# B&R Automation Studio project NAEUL004C00R13L518F00 (part 67)

#### Act_InitGlobal.st - Change By Project
```iecst
(** 2019-04-16 **)
ACTION Act_InitGlobal:

	(* Always Change If Project Change *)

	//Pass Data To Link

	p_bLinkNtParamMagConv1Prep ACCESS p_NtParamProjMag1ConvPrep;
	p_bLinkNtParamMagConv2Prep ACCESS p_NtParamProjMag2ConvPrep;
	p_bLinkNtParamMagConv3Prep ACCESS p_NtParamProjMag3ConvPrep;
	p_bLinkUSHermesABlkUS ACCESS p_USHermesABlkUS;
	p_bLinkUSHermesBBlkUS ACCESS p_USHermesBBlkUS;
	p_bLinkFollower1USAllow ACCESS p_Follower1USAllow;
	p_bLinkFollower2DSAllow ACCESS p_Follower2DSAllow;
	p_bLinkProjLifterMagPlatform ACCESS p_NtParamProjLifterMagPlatform;
	p_bLinkDIPshrAntiJamSen ACCESS p_DIPshrAntiJamSen;
	p_bLinkCurtainSen ACCESS p_DICurtainSen;
	p_bLinkPshrRetSen ACCESS p_DIPusherRetRS;

	p_diBuffer1NxtLoadSlt ACCESS p_Buffer1NxtLoadSlt;
	p_diBuffer2NxtLoadSlt ACCESS p_Buffer2NxtLoadSlt;
	p_diBuffer3NxtLoadSlt ACCESS p_Buffer3NxtLoadSlt;

	p_diMinSlt ACCESS p_ProdRcpCurrRcp1MinSltValue;
	p_diMaxSlt ACCESS p_ProdRcpCurrRcp1MaxSltValue;

	p_bTopToBtm ACCESS p_ProdRcpCurrRcp1TopToBtm;

	p_bLinkMcParamMagWidthChkDis ACCESS p_McParamMagWidthChkDis;

	//p_bMagWidthChkDis
	p_sLinkProdRcpCurrRcp1Nm ACCESS p_ProdRcpCurrRcp1Nm;
	p_diLinkProdRcpCurrRcp1Pitch ACCESS p_ProdRcpCurrRcp1Pitch;
	p_sLinkMagRcpCurrRcpNm ACCESS p_MagRcpCurrRcpNm;

	//Pass Data To Internal Use
	p_udiRstErr ACCESS p_RstErrReset;
	p_bRun ACCESS p_OpsRun;
	p_bStop ACCESS p_OpsStop;
	p_bStep ACCESS p_OpsStep;

	p_tShutterWaitTmr ACCESS p_NtParamShutterWaitTmr;
	p_bCurtainSenPrep ACCESS p_NtParamCurtainSenPrep;

	p_sProgNm ACCESS p_NtParamOpsTravLifULProgNm;
	p_bNtSettingsLoadDone ACCESS p_StartupNtSettingsLoadDone;

	p_eULMag ACCESS p_NtParamProjMag;
	p_bInShutDis ACCESS p_McParamInShutterDis;

	p_eUSCommMod1 ACCESS p_McParamUSCommAMod;
	p_eUSCommMod2 ACCESS p_McParamUSCommBMod;

	p_eUSSMEMAStat1 ACCESS p_USSMEMAAStat;
	p_eUSSMEMAStatus1 ACCESS p_USSMEMAAStatus;
	p_bUSSMEMAUSRdy1 ACCESS p_USSMEMAAUSRdy;
	p_bUSSMEMAGdBrdRdy1 ACCESS p_USSMEMAAUSGdBrdRdy;
	p_bUSSMEMATransporting1 ACCESS p_USSMEMAATransporting;
	p_bUSSMEMAConvStart1 ACCESS p_USSMEMAAConvStart;
	p_bUSSMEMAConvStop1 ACCESS p_USSMEMAAConvStop;

	p_eUSSMEMAStat2 ACCESS p_USSMEMABStat;
	p_eUSSMEMAStatus2 ACCESS p_USSMEMABStatus;
	p_bUSSMEMAUSRdy2 ACCESS p_USSMEMABUSRdy;
	p_bUSSMEMAGdBrdRdy2 ACCESS p_USSMEMABUSGdBrdRdy;
	p_bUSSMEMATransporting2 ACCESS p_USSMEMABTransporting;
	p_bUSSMEMAConvStart2 ACCESS p_USSMEMABConvStart;
	p_bUSSMEMAConvStop2 ACCESS p_USSMEMABConvStop;

	p_eDSSMEMAStat1 ACCESS p_DSSMEMA1Stat;
	p_eDSSMEMAStatus1 ACCESS p_DSSMEMA1Status;
	p_bDSSMEMADSRdy1 ACCESS p_DSSMEMA1DSRdy;
	p_bDSSMEMAConvStart1 ACCESS p_DSSMEMA1ConvStart;

	p_eDSSMEMAStat2 ACCESS p_DSSMEMA2Stat;
	p_eDSSMEMAStatus2 ACCESS p_DSSMEMA2Status;
	p_bDSSMEMADSRdy2 ACCESS p_DSSMEMA2DSRdy;
	p_bDSSMEMAConvStart2 ACCESS p_DSSMEMA2ConvStart;

	p_eDSSMEMAStat3 ACCESS p_DSSMEMA3Stat;
	p_eDSSMEMAStatus3 ACCESS p_DSSMEMA3Status;
	p_bDSSMEMADSRdy3 ACCESS p_DSSMEMA3DSRdy;
	p_bDSSMEMAConvStart3 ACCESS p_DSSMEMA3ConvStart;

	p_bUSHermesUSRdy1 ACCESS p_USHermesAUSRdy;
	p_bUSHermesUSGdRdy1 ACCESS p_USHermesAUSGdRdy;
	p_bUSHermesTransporting1 ACCESS p_USHermesATransporting;
	p_bUSHermesStopTransport1 ACCESS p_USHermesAStopTransport;

	p_bUSHermesUSRdy2 ACCESS p_USHermesBUSRdy;
	p_bUSHermesUSGdRdy2 ACCESS p_USHermesBUSGdRdy;
	p_bUSHermesTransporting2 ACCESS p_USHermesBTransporting;
	p_bUSHermesStopTransport2 ACCESS p_USHermesBStopTransport;

	p_eConvStat ACCESS p_PshrConvStat;
	p_eConvStatus ACCESS p_PshrConvStatus;
	p_eConvDir ACCESS p_NtParamProjConvDir;
	p_bConvHvBrd ACCESS p_PshrConvHvBrd;
	p_bConvGdBrd ACCESS p_PshrConvGdBrd;

	p_eAWStat ACCESS p_AWOpenStat;
	p_eAWStatus ACCESS p_AWOpenStatus;
	p_bAWWidthPosDiff ACCESS p_AWOpenWidthPosDiff;

	p_eTravStat ACCESS p_TravStat;
	p_eTravStatus ACCESS p_TravStatus;

//	p_eLifStat ACCESS p_LifterBtmStat;
//	p_eLifStatus ACCESS p_LifterBtmStatus;

	p_eInletPneuStat ACCESS p_Pneu2SenInShutterStat;
	p_eInletPneuStatus ACCESS p_Pneu2SenInShutterStatus;
	p_bInletPneuCls ACCESS p_Pneu2SenInShutterExtended;

	p_eOutletPneuStat ACCESS p_Pneu2SenOutShutterStat;
	p_eOutletPneuStatus ACCESS p_Pneu2SenOutShutterStatus;

	p_eOutletPneuStat2 ACCESS p_Pneu2SenOutShutterStat2;
	p_eOutletPneuStatus2 ACCESS p_Pneu2SenOutShutterStatus2;

	p_eOutletPneuStat3 ACCESS p_Pneu2SenOutShutterStat3;
	p_eOutletPneuStatus3 ACCESS p_Pneu2SenOutShutterStatus3;

	p_eStopperStat1 ACCESS p_PneuNoSenStopperAStat;
	p_eStopperStatus1 ACCESS p_PneuNoSenStopperAStatus;
	p_bStopperBlk1 ACCESS p_PneuNoSenStopperAExtended;

	p_eStopperStat2 ACCESS p_PneuNoSenStopperBStat;
	p_eStopperStatus2 ACCESS p_PneuNoSenStopperBStatus;
	p_bStopperBlk2 ACCESS p_PneuNoSenStopperBExtended;

	p_eStopperStat3 ACCESS p_PneuNoSenStopperCStat;
	p_eStopperStatus3 ACCESS p_PneuNoSenStopperCStatus;
	p_bStopperBlk3 ACCESS p_PneuNoSenStopperCExtended;

	p_bConvLftSen ACCESS p_DIConvLftSen;
	p_bConvMidSen ACCESS p_DIConvMidSen;
	p_bConvRgtSen ACCESS p_DIConvRgtSen;
	p_bConvClrSen ACCESS p_DIConvClrSen;
	p_bConvLineAInletSen ACCESS p_DIConvLineAInletSen;
	p_bConvLineBInletSen ACCESS p_DIConvLineBInletSen;

	p_bBufferMagPresent1 ACCESS p_Buffer1MagPresent;
	p_bBufferMagPresent2 ACCESS p_Buffer2MagPresent;
	p_bBufferMagPresent3 ACCESS p_Buffer3MagPresent;

	p_bBufferMagDet1 ACCESS p_DIMagPresentSen1;
	p_bBufferMagDet2 ACCESS p_DIMagPresentSen2;
	p_bBufferMagDet3 ACCESS p_DIMagPresentSen3;

	p_tyBufferStat1 ACCESS p_Buffer1BffrStat;
	p_tyBufferStat2 ACCESS p_Buffer2BffrStat;
	p_tyBufferStat3 ACCESS p_Buffer3BffrStat;

	p_bTravAPosDiff ACCESS p_TravAPosDiff;
	p_bTravBPosDiff ACCESS p_TravBPosDiff;
	p_bTravPosDiff ACCESS p_TravPosDiff;
//	p_bLifterBtmPosDiff ACCESS p_LifterBtmPosDiff;
//	p_bLifterAPosDiff ACCESS p_LifterBtmAPosDiff;
//	p_bLifterBPosDiff ACCESS p_LifterBtmBPosDiff;

	p_bDIInShutterOpenRS ACCESS p_DIInShutterOpenRS;
	p_bDIInShutterCloseRS ACCESS p_DIInShutterCloseRS;
	p_bDIPusherExtRS ACCESS p_DIPusherExtRS;
	p_bDIPusherRetRS ACCESS p_DIPusherRetRS;
	p_bDIOutShutterOpenRS ACCESS p_DIOutShutterOpenRS;
	p_bDIOutShutterCloseRS ACCESS p_DIOutShutterCloseRS;
	p_bDIOutShutterOpenRS2 ACCESS p_DIOutShutterOpenRS2;
	p_bDIOutShutterCloseRS2 ACCESS p_DIOutShutterCloseRS2;
	p_bDIOutShutterOpenRS3 ACCESS p_DIOutShutterOpenRS3;
	p_bDIOutShutterCloseRS3 ACCESS p_DIOutShutterCloseRS3;
	p_bPshrConvPshrRetracted ACCESS p_PshrConvPshrRetracted;

	p_bMagWidthChkSenOn ACCESS p_DIMagWidthChkSen;

	p_eAWPushOrPullerStat ACCESS p_AWPushOrPullerStat;
	p_eAWPushOrPullerStatus ACCESS p_AWPushOrPullerStatus;
	p_bAWPushOrPullerWidthPosDiff ACCESS p_AWPushOrPullerPosDiff ;

	p_dtBufferMagPresentTm1 ACCESS p_Buffer1MagPresentTm;
	p_dtBufferMagPresentTm2 ACCESS p_Buffer2MagPresentTm;
	p_dtBufferMagPresentTm3 ACCESS p_Buffer3MagPresentTm;

	p_diProdRcpCurrRcp1Width ACCESS p_ProdRcpCurrRcp1Width;
	p_diProdRcpCurrRcp2Width ACCESS p_ProdRcpCurrRcp2Width;

	p_bCurtainSenPB ACCESS p_DICurtainSenPB;

	//	p_bScanEn ACCESS p_NtParamProjScanPrep; 		//Scanner
	p_bTopScannerEn ACCESS p_McParamTopScannerEn;
	p_bBtmScannerEn ACCESS p_McParamBtmScannerEn;

	p_eTCPTopStat ACCESS p_TCPTopStat;
	p_eTCPTopStatus ACCESS p_TCPTopStatus;
	p_sTopMsgRd ACCESS p_TCPTopFullMsgRd;

	p_eTCPBtmStat ACCESS p_TCPBtmStat;
	p_eTCPBtmStatus ACCESS p_TCPBtmStatus;
	p_sBtmMsgRd ACCESS p_TCPBtmFullMsgRd;
	p_bOpConPrep ACCESS p_NtParamProjOpConPrep;
	p_tyPartReceiveRetCode ACCESS p_OpConPartRcvRetCode;
	p_tyOpConPlcGrabRcvCode ACCESS p_OpConPlcGrabRcvCode;

	p_bOpsMagConvUL1UnclmpDone ACCESS p_OpsMagConvUL1UnclmpDone; // Access From Mag Conv UL 1,2,3
	p_bOpsMagConvUL2UnclmpDone ACCESS p_OpsMagConvUL2UnclmpDone;
	p_bOpsMagConvUL3UnclmpDone ACCESS p_OpsMagConvUL3UnclmpDone;

	p_bNtParamProjOutletShutPrep ACCESS p_NtParamProjOutletShutPrep;
	p_bNtParamProjOutletShut2Prep ACCESS p_NtParamProjOutletShut2Prep;
	p_bNtParamProjOutletShut3Prep ACCESS p_NtParamProjOutletShut3Prep;

	p_bAutoRcpTravWidthDiffBlk ACCESS p_AutoRcpbTravWidthDiffblk;

	p_bNtParamAutoRcpPrep ACCESS p_NtParamAutoRcpPrep;
	p_bMcParamAutoRcpDis  ACCESS p_McParamAutoRcpDisable;
	p_eNtParamAutoRcpPrecededBy ACCESS p_NtParamAutoRcpPrecededBy;
	//udiPosallow Go
	//p_udiOpsUSPosAllwGo ACCESS p_OpsUSPosAllwGo;
	//p_udiOpsDSPosAllwGo ACCESS p_OpsDSPosAllwGo;

	p_eCustomerReq ACCESS p_NtParamCustomerReq;
	//Inlet stopper
	p_bStopperUnBlkCtrl ACCESS p_InletStopperRetCtrl;
	p_eInletStopperStatus ACCESS p_InletStopperStatus;
	p_eInletStopperStat ACCESS p_InletStopperStat;
	p_bInletStopperPrep ACCESS p_NtParamProjInletStopperPrep;
	p_bDIInletStopperASen ACCESS p_DIInletStopperASen;
	p_diMcParamInStprExtDelayTm ACCESS p_McParamInStopperExtDelayTm;
	//OpCon
	p_bLinkOpConEn ACCESS p_McParamOpConEn;
	p_sTopBtmBarcode ACCESS p_USHermesATopBtmBarcode; //receive bc by hermes
	p_MCUL1StepPLCGrab ACCESS p_OpsMagConvUL1StepPLCGrab; //for opcon plcGrab
	p_MCUL2StepPLCGrab ACCESS p_OpsMagConvUL2StepPLCGrab;
	p_MCUL3StepPLCGrab ACCESS p_OpsMagConvUL3StepPLCGrab;
	p_bMagPresentSen1 ACCESS p_DIMagPresentSen1;
	p_bMagPresentSen2 ACCESS p_DIMagPresentSen2;
	p_bMagPresentSen3 ACCESS p_DIMagPresentSen3;
	//DMC Scanner
	p_tyNtParamDISettings ACCESS p_NtParamDISettings;
	p_tyNtParamDOSettings ACCESS p_NtParamDOSettings;
	p_bDIPCBScanComplSig ACCESS p_DIPCBScanComplSig;
	//Auto Bypass Curtain
	p_bRlsMag1 ACCESS p_UIRlsMag1 ;
	p_bRlsMag2 ACCESS p_UIRlsMag2;
	p_bRlsMag3 ACCESS p_UIRlsMag3;
	//Pusher Ret to Slow Sensor ,start traverse
	p_bPshrConvPshrRetSlwSen ACCESS p_PshrConvPshrRetAllwTrav;
	p_bMcParamDMCScannerEn ACCESS p_McParamDMCScannerEn;
	p_diMcParamDMCScanResponseTO ACCESS p_McParamDMCScanWriteTO;
	(* Always Change If Project Change *)
	//added
	p_iLifterSltMoved ACCESS p_LifterBtmMovedSlt;
END_ACTION
```

#### InputRef_Link.var - Change By Project
```iecst
(*2018-12-11*)
(**)
(*External Data*)
VAR
	p_usiLinkProdRcpCurrRcpMcMod : REFERENCE TO USINT;
	p_bLinkNtParamMagConv1Prep : REFERENCE TO USINT;
	p_bLinkNtParamMagConv2Prep : REFERENCE TO USINT;
	p_bLinkNtParamMagConv3Prep : REFERENCE TO USINT;
	p_bLinkUSHermesABlkUS : REFERENCE TO BOOL;
	p_bLinkUSHermesBBlkUS : REFERENCE TO BOOL;
	p_bLinkFollower1USAllow : REFERENCE TO BOOL;
	p_bLinkFollower2DSAllow : REFERENCE TO BOOL;
	p_bLinkProjLifterMagPlatform : REFERENCE TO BOOL;
	p_bLinkDIPshrAntiJamSen : REFERENCE TO BOOL;
	p_bLinkCurtainSen : REFERENCE TO BOOL;
	p_bLinkPshrRetSen : REFERENCE TO BOOL;
	p_diBuffer1NxtLoadSlt : REFERENCE TO DINT;
	p_diBuffer2NxtLoadSlt : REFERENCE TO DINT;
	p_diBuffer3NxtLoadSlt : REFERENCE TO DINT;
	p_diMinSlt : REFERENCE TO DINT;
	p_diMaxSlt : REFERENCE TO DINT;
	p_bTopToBtm : REFERENCE TO BOOL;
	p_bLinkMcParamMagWidthChkDis : REFERENCE TO BOOL;
	p_bMagWidthChkDis : REFERENCE TO BOOL;
	bMagWidthChkTravMov : BOOL;
	bMagWidthChk : BOOL;
	usiMagWidthChkStep : INT := 10;
	bTravGoToChkPt : BOOL;
	bShut1Closed : BOOL;
	bShut2Closed : BOOL;
	bShut3Closed : BOOL;
	p_bOpsMagConvUL1UnclmpDone : REFERENCE TO BOOL;
	p_bOpsMagConvUL2UnclmpDone : REFERENCE TO BOOL;
	p_bOpsMagConvUL3UnclmpDone : REFERENCE TO BOOL;
	p_bNtParamProjOutletShutPrep : REFERENCE TO BOOL;
	p_bNtParamProjOutletShut2Prep : REFERENCE TO BOOL;
	p_bNtParamProjOutletShut3Prep : REFERENCE TO BOOL;
	p_bAutoRcpTravWidthDiffBlk : REFERENCE TO BOOL;
	p_bNtParamAutoRcpPrep : REFERENCE TO BOOL;
	p_bMcParamAutoRcpDis : REFERENCE TO BOOL;
	p_eNtParamAutoRcpPrecededBy : REFERENCE TO eAutoRcpPreceded;
	p_eCustomerReq : REFERENCE TO eCustomer;
END_VAR
(*inlet stopper*)
VAR
	p_bInletStopperPrep : REFERENCE TO BOOL;
	p_bStopperUnBlkCtrl : REFERENCE TO BOOL;
	p_eInletStopperStat : REFERENCE TO ePneuAction;
	p_eInletStopperStatus : REFERENCE TO eFBStatus;
	p_bDIInletStopperASen : REFERENCE TO BOOL;
	p_diMcParamInStprExtDelayTm : REFERENCE TO DINT;
END_VAR
(*Ops AllwGo*)
VAR
	p_udiOpsUSPosAllwGo : REFERENCE TO UDINT;
	p_udiOpsDSPosAllwGo : REFERENCE TO UDINT;
END_VAR
(*AutoBypass Curtain*)
VAR
	p_bRlsMag1 : REFERENCE TO BOOL;
	p_bRlsMag2 : REFERENCE TO BOOL;
	p_bRlsMag3 : REFERENCE TO BOOL;
END_VAR
(*pusher react slow then traverse*)
VAR
	p_bPshrConvPshrRetSlwSen : REFERENCE TO BOOL;
	p_bMcParamDMCScannerEn : REFERENCE TO BOOL;
	p_iLifterSltMoved : REFERENCE TO INT;
	p_diMcParamDMCScanResponseTO : REFERENCE TO DINT;
END_VAR
(*opcon*)
VAR
	p_bLinkOpConEn : REFERENCE TO BOOL;
	p_sTopBtmBarcode : REFERENCE TO ARRAY[0..1] OF STRING[254];
	p_MCUL1StepPLCGrab : REFERENCE TO BOOL;
	p_MCUL2StepPLCGrab : REFERENCE TO BOOL;
	p_MCUL3StepPLCGrab : REFERENCE TO BOOL;
	p_bMagPresentSen1 : REFERENCE TO BOOL;
	p_bMagPresentSen2 : REFERENCE TO BOOL;
	p_bMagPresentSen3 : REFERENCE TO BOOL;
	p_bPLCGrabPic : REFERENCE TO BOOL;
	p_bDIPCBScanComplSig : REFERENCE TO BOOL;
	p_tyNtParamDOSettings : REFERENCE TO tyDigitalOutputSettings;
	p_tyNtParamDISettings : REFERENCE TO tyDigitalInputSettings;
END_VAR
(*for part process*)
VAR
	p_sLinkProdRcpCurrRcp1Nm : REFERENCE TO STRING[254];
	p_diLinkProdRcpCurrRcp1Pitch : REFERENCE TO DINT;
	p_sLinkMagRcpCurrRcpNm : REFERENCE TO STRING[30];
END_VAR
```

#### Act_LinkEn.st - Change By Project
```iecst
(** 2019-01-11 **)
ACTION Act_LinkEn:

	//Link bPrep, bEn & bDis
	p_bScanEn := p_bTopScannerEn OR p_bBtmScannerEn;
END_ACTION
```

#### Act_Link.st - Change By Project
```iecst
(** 2018-12-11 **)
ACTION Act_Link:
	//MagWidth Disable and Prep
	p_bMagWidthChkDis := NOT(p_tyNtParamDISettings.diUSWidthChkSen>0) OR p_bLinkMcParamMagWidthChkDis;
	//Disable AutoRcp
	//Upstream Allow
	IF p_bNtParamAutoRcpPrep AND NOT(p_bMcParamAutoRcpDis) THEN
		IF p_eNtParamAutoRcpPrecededBy = PrecededBySelf THEN
			p_usiLinkProdRcpCurrRcpMcMod ACCESS p_ProdRcpCurrRcp0McMod; //take respective Rcp
			p_bUSAllow := p_bAutoRcpTravWidthDiffBlk = FALSE;
		ELSIF p_eNtParamAutoRcpPrecededBy = PrecededByF1 THEN
			p_usiLinkProdRcpCurrRcpMcMod ACCESS p_ProdRcpCurrRcp1McMod;
			p_bUSAllow	:= p_bLinkFollower1USAllow AND p_bLinkUSHermesABlkUS = FALSE AND p_bLinkUSHermesBBlkUS = FALSE;
		END_IF
	ELSE
		p_usiLinkProdRcpCurrRcpMcMod ACCESS p_ProdRcpCurrRcp1McMod;
		p_bUSAllow	:= p_bLinkFollower1USAllow AND p_bLinkUSHermesABlkUS = FALSE AND p_bLinkUSHermesBBlkUS = FALSE;// AND p_bAutoRcpTravWidthDiffBlk = FALSE;// AND p_diProdRcpCurrRcp1Width = p_diProdRcpCurrRcp2Width;
	END_IF

	p_eULMod	:= USINT_TO_UDINT(p_usiLinkProdRcpCurrRcpMcMod);

	p_bPneuUnclmpFBDone := p_bOpsMagConvUL1UnclmpDone OR p_bOpsMagConvUL2UnclmpDone OR p_bOpsMagConvUL3UnclmpDone;

	CASE p_eULMod OF
		ULModUnloadFrontLnA, ULModUnloadRearLnB, ULModUnloadDualLnAB:
			bBypsGdBadBrd	:= TRUE;
		ULModRejFrontLnA, ULModRejFrontLnARev, ULModRejRearLnB, ULModRejRearLnBRev, ULModRejDualLnA, ULModRejDualLnB:
			bBypsGdBadBrd	:= FALSE;
	END_CASE

	IF p_bLinkProjLifterMagPlatform = FALSE THEN
		p_bMagTransferBrd1 ACCESS p_OpsMagConvUL1MagBffrAvl;
		p_bMagTransferBrd2 ACCESS p_OpsMagConvUL2MagBffrAvl;
		p_bMagTransferBrd3 ACCESS p_OpsMagConvUL3MagBffrAvl;
	ELSE
		p_bMagTransferBrd1 ACCESS p_DSSMEMA1DSRdy;
		p_bMagTransferBrd2 ACCESS p_DSSMEMA2DSRdy;
		p_bMagTransferBrd3 ACCESS p_DSSMEMA3DSRdy;
	END_IF

	//	p_bDSAllow	:= p_bLinkFollower2DSAllow;

	IF p_bLinkProjLifterMagPlatform = FALSE THEN
		p_eLifStat ACCESS p_LifterBtmStat;
		p_eLifStatus ACCESS p_LifterBtmStatus;
		p_bLifterBtmPosDiff ACCESS p_LifterBtmPosDiff;
		p_bLifterAPosDiff ACCESS p_LifterBtmAPosDiff;
		p_bLifterBPosDiff ACCESS p_LifterBtmBPosDiff;
	ELSIF p_bLinkProjLifterMagPlatform  AND p_bRun THEN
		p_eLifStat := eLifAct;
		p_eLifStatus := Done; //bi-dir
		p_bLifterBtmPosDiff ACCESS ADR(bLifterBtmPosDiff);
		p_bLifterAPosDiff ACCESS ADR(bLifterAPosDiff);
		p_bLifterBPosDiff ACCESS ADR(bLifterBPosDiff);
	END_IF

	IF p_bRun AND p_bLinkDIPshrAntiJamSen = FALSE THEN
		eStatus		:= Error;
		udiStatus	:= 10005;
	END_IF

	//Bypass Curtain Sensor PB Pressed
	IF p_bRun THEN
		IF EDGENEG(p_bRlsMag1 OR p_bRlsMag2 OR p_bRlsMag3) THEN
			bBypCurtainSenPB 		:= TRUE;
			bBypCurtainSensorPBLED	:= TRUE;
		ELSIF EDGENEG (p_bCurtainSenPB) THEN
			IF bBypCurtainSenPB 		= TRUE THEN
				bBypCurtainSenPB		:= FALSE;
				bBypCurtainSensorPBLED	:= FALSE;
				bBypCurtainSenCtrl		:= FALSE;
				bWait					:= FALSE;
			ELSE
				bBypCurtainSenPB 		:= TRUE;
				bBypCurtainSensorPBLED	:= TRUE;
			END_IF
		END_IF
	ELSE
		bBypCurtainSenPB		:= FALSE;
		bBypCurtainSensorPBLED	:= FALSE;
		bBypCurtainSenCtrl		:= FALSE;
	END_IF

	//Run & Initializing Done Bypass the Curtain Sensor
	IF bBypCurtainSenPB AND p_eTravStatus <> Busy AND p_eLifStatus <> Busy AND bWait = FALSE THEN
		bWait 	:= TRUE;
	END_IF

	IF p_bRun AND bOpsInitDone AND bBypCurtainSenPB AND bWait THEN
		bBypCurtainSenCtrl		:= TRUE;
	ELSE
		bBypCurtainSenCtrl		:= FALSE;
	END_IF

	// BypCurtainSensorPBLED
	IF  (bBypCurtainSenPB = TRUE) AND (bBypCurtainSenCtrl = TRUE) THEN
		bBypCurtainSensorPBLED := TRUE;
		fbBypCurtainPBLEDBlinkTm(IN := FALSE);
	ELSIF (bBypCurtainSenPB = TRUE) AND (bBypCurtainSenCtrl = FALSE) THEN
		fbBypCurtainPBLEDBlinkTm(IN := TRUE);
		IF fbBypCurtainPBLEDBlinkTm.Q = TRUE THEN
			fbBypCurtainPBLEDBlinkTm(IN := FALSE);
			IF bBypCurtainSensorPBLED = FALSE THEN
				bBypCurtainSensorPBLED := TRUE;
			ELSE
				bBypCurtainSensorPBLED := FALSE;
			END_IF
		END_IF
	ELSE
		bBypCurtainSensorPBLED := FALSE;
		fbBypCurtainPBLEDBlinkTm(IN := FALSE);
	END_IF

	//for inlet outlet sensing
	fb2SenTm(IN:= p_bConvRgtSen = TRUE AND p_bConvLftSen= TRUE, PT:= T#500ms);
	IF fb2SenTm.Q = TRUE THEN
		eStatus := Error;
		udiStatus := 10009; //'Inlet and outlet same time sensing error'
	END_IF

//	fbRstCurtain(IN := bBypCurtainSenCtrl); //Auto Reset when the bypass curtain Sen is On more than 1 min.
//
//	IF p_bLinkCurtainSen AND fbRstCurtain.Q THEN
//		bBypCurtainSenCtrl		:= FALSE;
//		bBypCurtainSenPB		:= FALSE;
//		bBypCurtainSensorPBLED	:= FALSE;
//	END_IF

//Machine Paused and Bypass Curtain Sensor
//	IF bBypCurtainSenPB THEN
//
//		eOutletPneuAct	:= PneuActExt;
//		eOutletPneuAct2	:= PneuActExt;
//		eOutletPneuAct3	:= PneuActExt;
//
//		IF (p_eOutletPneuStatus = Done AND p_eOutletPneuStat = PneuActExt) AND (p_eOutletPneuStatus2 = Done AND p_eOutletPneuStat2 = PneuActExt) AND (p_eOutletPneuStatus3 = Done AND p_eOutletPneuStat3 = PneuActExt) THEN
//			eOutletPneuAct	:= PneuActIdle;
//			eOutletPneuAct2	:= PneuActIdle;
//			eOutletPneuAct2	:= PneuActIdle;
//			bBypCurtainSenCtrl := TRUE;
//		END_IF
//	END_IF

END_ACTION
```

#### Act_InitLocal.st - Do Not Change!!!
```iecst
(** 2019-04-16 **)
ACTION Act_InitLocal:

	//Input Reference Link To Local Variable
	p_udiRstErr ACCESS ADR(udiRstErr);
	p_bEn ACCESS ADR(bEn);
	p_bDis ACCESS ADR(bDis);
	p_bRun ACCESS ADR(bRun);
	p_bStop ACCESS ADR(bStop);
	p_bStep ACCESS ADR(bStep);

	p_sProgNm ACCESS ADR(sProgNm);
	p_bNtSettingsLoadDone ACCESS ADR(bNtSettingsLoadDone);

	p_eULMod ACCESS ADR(eULMode);
	p_eULMag ACCESS ADR(eULMagazine);
	p_bNonBffrMod ACCESS ADR(bNonBffrMod);
	p_bBypsGdBadBrd ACCESS ADR(bBypsGdBadBrd);
	p_bUSAllow ACCESS ADR(bUSAllow);
	p_bDSAllow ACCESS ADR(bDSAllow);

	p_eUSCommMod1 ACCESS ADR(eUSCommMod1);
	p_eUSCommMod2 ACCESS ADR(eUSCommMod2);
	p_eUSCommMod3 ACCESS ADR(eUSCommMod3);
	p_eDSCommMod1 ACCESS ADR(eDSCommMod1);
	p_eDSCommMod2 ACCESS ADR(eDSCommMod2);
	p_eDSCommMod3 ACCESS ADR(eDSCommMod3);

	p_eUSSMEMAStat1 ACCESS ADR(eUSSMEMAStat1);
	p_eUSSMEMAStatus1 ACCESS ADR(eUSSMEMAStatus1);
	p_bUSSMEMAUSRdy1 ACCESS ADR(bUSSMEMAUSRdy1);
	p_bUSSMEMAGdBrdRdy1 ACCESS ADR(bUSSMEMAGdBrdRdy1);
	p_bUSSMEMATransporting1 ACCESS ADR(bUSSMEMATransporting1);
	p_bUSSMEMAConvStart1 ACCESS ADR(bUSSMEMAConvStart1);
	p_bUSSMEMAConvStop1 ACCESS ADR(bUSSMEMAConvStop1);

	p_eUSSMEMAStat2 ACCESS ADR(eUSSMEMAStat2);
	p_eUSSMEMAStatus2 ACCESS ADR(eUSSMEMAStatus2);
	p_bUSSMEMAUSRdy2 ACCESS ADR(bUSSMEMAUSRdy2);
	p_bUSSMEMAGdBrdRdy2 ACCESS ADR(bUSSMEMAGdBrdRdy2);
	p_bUSSMEMATransporting2 ACCESS ADR(bUSSMEMATransporting2);
	p_bUSSMEMAConvStart2 ACCESS ADR(bUSSMEMAConvStart2);
	p_bUSSMEMAConvStop2 ACCESS ADR(bUSSMEMAConvStop2);

	p_eUSSMEMAStat3 ACCESS ADR(eUSSMEMAStat3);
	p_eUSSMEMAStatus3 ACCESS ADR(eUSSMEMAStatus3);
	p_bUSSMEMAUSRdy3 ACCESS ADR(bUSSMEMAUSRdy3);
	p_bUSSMEMAGdBrdRdy3 ACCESS ADR(bUSSMEMAGdBrdRdy3);
	p_bUSSMEMATransporting3 ACCESS ADR(bUSSMEMATransporting3);
	p_bUSSMEMAConvStart3 ACCESS ADR(bUSSMEMAConvStart3);
	p_bUSSMEMAConvStop3 ACCESS ADR(bUSSMEMAConvStop3);

	p_eDSSMEMAStat1 ACCESS ADR(eDSSMEMAStat1);
	p_eDSSMEMAStatus1 ACCESS ADR(eDSSMEMAStatus1);
	p_bDSSMEMADSRdy1 ACCESS ADR(bDSSMEMADSRdy1);
	p_bDSSMEMAConvStart1 ACCESS ADR(bDSSMEMAConvStart1);

	p_eDSSMEMAStat2 ACCESS ADR(eDSSMEMAStat2);
	p_eDSSMEMAStatus2 ACCESS ADR(eDSSMEMAStatus2);
	p_bDSSMEMADSRdy2 ACCESS ADR(bDSSMEMADSRdy2);
	p_bDSSMEMAConvStart2 ACCESS ADR(bDSSMEMAConvStart2);

	p_eDSSMEMAStat3 ACCESS ADR(eDSSMEMAStat3);
	p_eDSSMEMAStatus3 ACCESS ADR(eDSSMEMAStatus3);
	p_bDSSMEMADSRdy3 ACCESS ADR(bDSSMEMADSRdy3);
	p_bDSSMEMAConvStart3 ACCESS ADR(bDSSMEMAConvStart3);

	p_bUSHermesUSRdy1 ACCESS ADR(bUSHermesUSRdy1);
	p_bUSHermesUSGdRdy1 ACCESS ADR(bUSHermesUSGdRdy1);
	p_bUSHermesTransporting1 ACCESS ADR(bUSHermesTransporting1);
	p_bUSHermesStopTransport1 ACCESS ADR(bUSHermesStopTransport1);

	p_bUSHermesUSRdy2 ACCESS ADR(bUSHermesUSRdy2);
	p_bUSHermesUSGdRdy2 ACCESS ADR(bUSHermesUSGdRdy2);
	p_bUSHermesTransporting2 ACCESS ADR(bUSHermesTransporting2);
	p_bUSHermesStopTransport2 ACCESS ADR(bUSHermesStopTransport2);

	p_bUSHermesUSRdy3 ACCESS ADR(bUSHermesUSRdy3);
	p_bUSHermesUSGdRdy3 ACCESS ADR(bUSHermesUSGdRdy3);
	p_bUSHermesTransporting3 ACCESS ADR(bUSHermesTransporting3);
	p_bUSHermesStopTransport3 ACCESS ADR(bUSHermesStopTransport3);

	p_bDSHermesDSRdy1 ACCESS ADR(bDSHermesDSRdy1);
	p_bDSHermesTransporting1 ACCESS ADR(bDSHermesTransporting1);
	p_bDSHermesStopTransport1 ACCESS ADR(bDSHermesStopTransport1);

	p_bDSHermesDSRdy2 ACCESS ADR(bDSHermesDSRdy2);
	p_bDSHermesTransporting2 ACCESS ADR(bDSHermesTransporting2);
	p_bDSHermesStopTransport2 ACCESS ADR(bDSHermesStopTransport2);

	p_bDSHermesDSRdy3 ACCESS ADR(bDSHermesDSRdy3);
	p_bDSHermesTransporting3 ACCESS ADR(bDSHermesTransporting3);
	p_bDSHermesStopTransport3 ACCESS ADR(bDSHermesStopTransport3);

	p_eConvStat	ACCESS ADR(eConvStat);
	p_eConvStatus ACCESS ADR(eConvStatus);
	p_eConvDir ACCESS ADR(eConvDirection);
	p_bConvHvBrd ACCESS ADR(bConvHvBrd);
	p_bConvGdBrd ACCESS ADR(bConvGdBrd);

	p_eAWStat ACCESS ADR(eAWStat);
	p_eAWStatus ACCESS ADR(eAWStatus);
	p_bAWWidthPosDiff ACCESS ADR(bAWWidthPosDiff);

	p_eTravStat ACCESS ADR(eTravStat);
	p_eTravStatus ACCESS ADR(eTravStatus);

	p_eLifStat ACCESS ADR(eLifStat);
	p_eLifStatus ACCESS ADR(eLifStatus);
	p_bLifterBtmPosDiff ACCESS ADR(bLifterBtmPosDiff);
	p_bLifterAPosDiff ACCESS ADR(bLifterAPosDiff);
	p_bLifterBPosDiff ACCESS ADR(bLifterBPosDiff);

	p_eInletPneuStat ACCESS ADR(eInletPneuStat);
	p_eInletPneuStatus ACCESS ADR(eInletPneuStatus);
	p_bInletPneuCls ACCESS ADR(bInletPneuCls);

	p_eOutletPneuStat ACCESS ADR(eOutletPneuStat);
	p_eOutletPneuStatus ACCESS ADR(eOutletPneuStatus);

	p_bConvLftSen ACCESS ADR(bConvLftSen);
	p_bConvRgtSen ACCESS ADR(bConvRgtSen);

	p_bMagTransferBrd1 ACCESS ADR(bMagTransferBrd1);
	p_bMagTransferBrd2 ACCESS ADR(bMagTransferBrd2);
	p_bMagTransferBrd3 ACCESS ADR(bMagTransferBrd3);
	p_bBufferMagPresent1 ACCESS ADR(bBufferMagPresent1);
	p_bBufferMagPresent2 ACCESS ADR(bBufferMagPresent2);
	p_bBufferMagPresent3 ACCESS ADR(bBufferMagPresent3);

	p_bPneuUnclmpFBDone ACCESS ADR(bPneuUnclmpFBDone);

	p_tShutterWaitTmr ACCESS ADR(tShutterWaitTmr);
	p_eNtParamProjMagBuffferActLoad	ACCESS ADR(eMagBuffferActLoad);

	p_bScanEn ACCESS ADR(bScanEn);
	p_eTCPTopStat ACCESS ADR(eTCPTopStat);
	p_eTCPTopStatus ACCESS ADR(eTCPTopStatus);
	p_sTopMsgRd ACCESS ADR(sTopMsgRd);
	p_eTCPBtmStat ACCESS ADR(eTCPBtmStat);
	p_eTCPBtmStatus ACCESS ADR(eTCPBtmStatus);
	p_sBtmMsgRd ACCESS ADR(sBtmMsgRd);

	p_bPass ACCESS ADR(bPass);
	p_tyPartReceiveRetCode ACCESS ADR(tyPartReceive);
	p_bPLCGrabPic ACCESS ADR (bPLCGrabPic);
	p_eLocalUSCommMod ACCESS ADR(eLocalUSCommMod);
	p_bMagWidthChkDis ACCESS ADR(bMagWidthChkDis);
END_ACTION
```

#### Act_Alarm.st - Do Not Change!!!
```iecst
(** 2019-03-25 **)
ACTION Act_Alarm:

	//Error
	IF EDGEPOS(eStatus = Error) THEN

		tyAlmData.sProgNm		:= p_sProgNm;
		tyAlmData.udiCode		:= udiStatus;
		tyAlmData.eSeverity		:= AlmSeverityError;
		tyAlmData.udiRunTime	:= tyAlmData.udiRunTime + 1;
		tyAlmData.bAlm			:= TRUE;
		tyAlmData.udiModuleNum  := udiModuleNum;
		g_sOpsTravLifULProgNm		:= p_sProgNm;

		//Get Error Message
		IF tyAlmData.udiCode < 10000 OR tyAlmData.udiCode > 10099 THEN
			tyAlmData.sAlmMsg	:= 'Unknown';
			tyAlmData.sRcyMsg	:= 'Unknown';
		ELSE
			tyAlmData.sAlmMsg	:= a_tyAlmText[tyAlmData.udiCode].sAlmText;
			tyAlmData.sRcyMsg	:= a_tyAlmText[tyAlmData.udiCode].sRcyText;
		END_IF

	ELSIF bRstErr AND (tyAlmData.udiCode <> 0) THEN

		tyAlmData.udiCode		:= 0;
		tyAlmData.eSeverity		:= AlmSeverityNA;
		tyAlmData.sAlmMsg		:= '';
		tyAlmData.sRcyMsg		:= '';
		tyAlmData.bAlm			:= FALSE;
	END_IF

END_ACTION
```

#### Package Logical/Operations/OpsTravLifUL/Sequence - Change By Project

#### Act_OpsInitial.st - Do Not Change!!!
```iecst
(** 2019-01-16 **)
ACTION Act_OpsInitial:

	eOpsStep		:= TravLifULStepNA;
	eGotoOpsStep	:= TravLifULStepInitConv;

	bInitConv		:= FALSE;
	bOpsInitDone	:= FALSE;
	bUSComm			:= FALSE;
	bEntBrd			:= FALSE;
	bDSComm			:= FALSE;
	bExitBrd		:= FALSE;

	usiMagWidthChkStep  := 0;
	bMagWidthChk		:= FALSE;
	bTravGoToChkPt		:= FALSE;

	bShut1Closed		:= FALSE;
	bShut2Closed		:= FALSE;
	bShut3Closed		:= FALSE;

END_ACTION
```

#### Act_OpsCommSig.st
```iecst
ACTION Act_OpsCommSig:
	IF bSelfTest = FALSE THEN
		//Upstream
		IF p_eUSCommMod1 = McSetCommModHermes THEN
			bLocalUSRdy1	:= p_bUSHermesUSRdy1;
			bLocalUSGdRdy1	:= p_bUSHermesUSGdRdy1;
		ELSE
			bLocalUSRdy1	:= p_bUSSMEMAUSRdy1;
			bLocalUSGdRdy1	:= p_bUSSMEMAGdBrdRdy1;
		END_IF

		IF p_eUSCommMod2 = McSetCommModHermes THEN
			bLocalUSRdy2	:= p_bUSHermesUSRdy2;
			bLocalUSGdRdy2	:= p_bUSHermesUSGdRdy2;
		ELSE
			bLocalUSRdy2	:= p_bUSSMEMAUSRdy2;
			bLocalUSGdRdy2	:= p_bUSSMEMAGdBrdRdy2;
		END_IF

		IF p_eUSCommMod3 = McSetCommModHermes THEN
			bLocalUSRdy3	:= p_bUSHermesUSRdy3;
			bLocalUSGdRdy3	:= p_bUSHermesUSGdRdy3;
		ELSE
			bLocalUSRdy3	:= p_bUSSMEMAUSRdy3;
			bLocalUSGdRdy3	:= p_bUSSMEMAGdBrdRdy3;
		END_IF

		//Downstream
		IF p_eDSCommMod1 = McSetCommModHermes THEN
			bLocalDSRdy1	:= p_bDSHermesDSRdy1;
		ELSE
			bLocalDSRdy1	:= p_bDSSMEMADSRdy1;
		END_IF

		IF p_eDSCommMod2 = McSetCommModHermes THEN
			bLocalDSRdy2	:= p_bDSHermesDSRdy2;
		ELSE
			bLocalDSRdy2	:= p_bDSSMEMADSRdy2;
		END_IF

		IF p_eDSCommMod3 = McSetCommModHermes THEN
			bLocalDSRdy3	:= p_bDSHermesDSRdy3;
		ELSE
			bLocalDSRdy3	:= p_bDSSMEMADSRdy3;
		END_IF

	ELSE
		IF eGotoOpsStep = TravLifULStepUSSigWait THEN

			bLocalUSRdy1 := TRUE;

		ELSIF eGotoOpsStep = TravLifULStepEntBrd AND p_bConvHvBrd THEN
			bLocalUSRdy1 := FALSE;
			bLocalUSRdy2 := FALSE;
			bLocalUSRdy3 := FALSE;
		END_IF
		//Downstream
		IF p_eDSCommMod1 = McSetCommModHermes THEN
			bLocalDSRdy1	:= p_bDSHermesDSRdy1;
		ELSE
			bLocalDSRdy1	:= p_bDSSMEMADSRdy1;
		END_IF

		IF p_eDSCommMod2 = McSetCommModHermes THEN
			bLocalDSRdy2	:= p_bDSHermesDSRdy2;
		ELSE
			bLocalDSRdy2	:= p_bDSSMEMADSRdy2;
		END_IF

		IF p_eDSCommMod3 = McSetCommModHermes THEN
			bLocalDSRdy3	:= p_bDSHermesDSRdy3;
		ELSE
			bLocalDSRdy3	:= p_bDSSMEMADSRdy3;
		END_IF
	END_IF
END_ACTION
```

#### Act_OpsStopper.st
```iecst
ACTION Act_OpsStopper:

	//Additional Script for Inlet Stopper

	IF eOpsStep <> TravLifULStepUSComm AND eOpsStep <> TravLifULStepInitConv AND  eOpsStep <>  TravLifULStepEntBrd AND eOpsStep <> TravLifULStepStopperRet THEN
		IF  p_bStopperUnBlkCtrl THEN// AND p_bDIInletStopperASen = FALSE THEN //(p_bAWWidthPosDiff OR NOT(p_bUSAllow)) AND
			eInletStopperAct	:= PneuActExt;
		END_IF
	END_IF
	IF eOpsStep = TravLifULStepUSComm  THEN
		IF p_bStopperUnBlkCtrl = FALSE AND (p_bLocalUSSMEMATransporting = TRUE OR p_bLocalUSHermesTransporting = TRUE) THEN //AND p_bDIInletStopperASen = TRUE THEN
			eInletStopperAct	:= PneuActRet;
		ELSIF p_bStopperUnBlkCtrl = TRUE AND (p_bLocalUSSMEMATransporting = FALSE AND p_bLocalUSHermesTransporting =  FALSE) THEN
			eInletStopperAct	:= PneuActExt;
		END_IF
	END_IF
	IF eOpsStep =  TravLifULStepInitConv OR eOpsStep =  TravLifULStepEntBrd THEN  //--> stopper sensor --> stopper --> inlet shutter --> inlet sensor
		IF EDGENEG(p_bDIInletStopperASen)  THEN
			bBrdOnStopperSen  := TRUE;
		END_IF
		fbInletStopperOffTim(IN := bBrdOnStopperSen,PT := DINT_TO_TIME(p_diMcParamInStprExtDelayTm) );

		IF p_bConvLftSen OR p_bConvRgtSen THEN
			bStopperBrdOnSen	:= TRUE;
		END_IF

		IF bStopperBrdOnSen   THEN
			IF NOT(p_bConvLftSen)   THEN
				eInletStopperAct	:= PneuActExt;
			END_IF
		END_IF
		IF bBrdOnStopperSen THEN
			IF fbInletStopperOffTim.Q THEN
				eInletStopperAct	:= PneuActExt;
			END_IF
		END_IF
	END_IF

	IF p_bStopperUnBlkCtrl THEN //retract
		IF p_eInletStopperStatus = Done AND p_eInletStopperStat = PneuActRet THEN
			eInletStopperAct	:= PneuActIdle;
		END_IF
	END_IF

	IF p_bStopperUnBlkCtrl = FALSE THEN	//exted
		IF p_eInletStopperStatus = Done AND p_eInletStopperStat = PneuActExt THEN
			eInletStopperAct	:= PneuActIdle;
		END_IF
		bStopperBrdOnSen	:= FALSE;
		bBrdOnStopperSen	:= FALSE;
		fbInletStopperOffTim(IN := FALSE);
	END_IF

END_ACTION
```

#### Act_OpsOpCon.st
```iecst
ACTION Act_OpsOpCon:
	//@@@@@@@@@@@@@@@@@@@@@@@@@@@@ opcon @@@@@@@@@@@@@@@@@@@@@@@@@@@@@@@@@@@@@@@@@@@@@@@@@@@@@@@@
	//intterupt condition
	p_bPass := p_tyPartReceiveRetCode.tyData.iReturnCode = 0;
	IF eGotoOpsStep = eOpsStep THEN
		CASE eOpsStep OF 	//Opcon step
			TravLifULStepScanDS: //SCAN MODE
				sStepTxt	:= 'Scanning In Progress';
				IF p_bConvHvBrd AND p_bConvRgtSen THEN
					eTCPTopAct := TCPActFullWriteReadUntilValid;
					eTCPBtmAct := TCPActFullWriteReadUntilValid;
				END_IF

				IF (p_eTCPTopStatus = Done AND p_eTCPTopStat = TCPActFullWriteReadUntilValid) OR
					(p_eTCPBtmStatus = Done AND p_eTCPBtmStat = TCPActFullWriteReadUntilValid) THEN
					IF p_sTopMsgRd = 'NOREAD$r$n' AND p_sBtmMsgRd = 'NOREAD$r$n'  THEN //2sec (config set from DLCode)
						eStatus		:= Error;
						udiStatus	:= 10006; // No Barcode Detected.
					ELSIF (p_sTopMsgRd = 'NOREAD$r$n' AND p_bBtmScannerEn = FALSE) OR (p_sBtmMsgRd = 'NOREAD$r$n' AND p_bTopScannerEn = FALSE) THEN
						eStatus		:= Error;
						udiStatus	:= 10006; // No Barcode Detected.
					ELSE // success scanned
						IF p_sTopMsgRd <> '' AND p_sTopMsgRd <> 'NOREAD$r$n' THEN
							//pass read data to opConXML.
							sBarcode := p_sTopMsgRd;

							eTCPTopAct := TCPActIdle_0;
							eTCPBtmAct := TCPActIdle_0;
							eGotoOpsStep := TravLifULStepWaitReturnCode;
						ELSIF p_sBtmMsgRd <> '' AND p_sBtmMsgRd <> 'NOREAD$r$n' THEN
							//pass read data to opConXML.
							sBarcode := p_sBtmMsgRd;

							eTCPTopAct := TCPActIdle_0;
							eTCPBtmAct := TCPActIdle_0;
							eGotoOpsStep := TravLifULStepWaitReturnCode;
						END_IF
					END_IF
				END_IF
				bPaused	:= p_bStop OR p_bStep;

			TravLifULStepHermesBCode:
				sStepTxt	:= 'Retrieve Barcode';
				bHermesBC := TRUE;
				IF p_sTopBtmBarcode[0] <> '' AND p_sTopBtmBarcode[0] <> 'NOREAD' THEN
					sBarcode 		:= p_sTopBtmBarcode[0];

					eGotoOpsStep  	:= TravLifULStepWaitReturnCode;
					p_tyPartReceiveRetCode.tyAvl.bReturnCode := FALSE;
				ELSIF p_sTopBtmBarcode[1] <> '' AND p_sTopBtmBarcode[1] <> 'NOREAD' THEN
					sBarcode 		:= p_sTopBtmBarcode[1];

					eGotoOpsStep 	:= TravLifULStepWaitReturnCode;
					p_tyPartReceiveRetCode.tyAvl.bReturnCode := FALSE;
				ELSE //both empty bc read
					eStatus		:= Error;
					udiStatus	:= 10006; // No Barcode Detected.
				END_IF
				bPaused	:= p_bStop OR p_bStep;

			TravLifULStepWaitReturnCode:
				sStepTxt	:= 'Wait Return Code';

				fbReturnCodeTO (IN:=TRUE); //10s
				IF p_bScanEn OR bHermesBC THEN
					IF p_bPass AND p_tyPartReceiveRetCode.tyAvl.bReturnCode THEN //ret 0
						eGotoOpsStep := TravLifULStepTravLifMov;
						fbReturnCodeTO (IN:=FALSE);
						p_sTopBtmBarcode[0] := '';
						p_sTopBtmBarcode[1] := '';
					ELSIF p_tyPartReceiveRetCode.tyAvl.bReturnCode AND
						(p_tyPartReceiveRetCode.tyData.iReturnCode = -1 OR p_tyPartReceiveRetCode.tyData.iReturnCode = -2) THEN
						eStatus		:= Error;
						udiStatus	:= 10008;  //change to reference to partRcv sTraceTxt
					ELSIF fbReturnCodeTO.Q THEN
						eStatus		:= Error;
						udiStatus	:= 10007; //Return Code Feedback Timeout.
					END_IF
				ELSE
					eGotoOpsStep := TravLifULStepTravLifMov;
				END_IF

				bPaused	:= p_bStop OR p_bStep;

			TravLifULStepMagChkReturnCode:
				sStepTxt	:= 'Magazine Verifing Standby Step';
				tyOpConMsgReq := OpConMsgTypeNA;
				fbReturnCodeTO (IN:=TRUE); //10s

				IF (p_tyOpConPlcGrabRcvCode.tyData.iReturnCode = 0) AND p_tyOpConPlcGrabRcvCode.tyAvl.bReturnCode THEN //ret 0
					eGotoOpsStep := TravLifULStepTravLifMov;
					bWaitMagChkRetCode := FALSE;
					fbReturnCodeTO (IN:=FALSE);
					p_tyOpConPlcGrabRcvCode.tyAvl.bReturnCode := FALSE;
				ELSIF p_tyOpConPlcGrabRcvCode.tyAvl.bReturnCode AND
					(p_tyOpConPlcGrabRcvCode.tyData.iReturnCode = -1 ) THEN
					eStatus		:= Error;
					udiStatus	:= 10010;  //change to reference to partRcv sTraceTxt
				ELSIF fbReturnCodeTO.Q THEN
					eStatus		:= Error;
					udiStatus	:= 10007; //Return Code Feedback Timeout.
				END_IF

		END_CASE
	END_IF
	//Reset Msg
	IF bJamStarted AND p_bConvHvBrd THEN
		bJamStarted := FALSE;
		tyOpConMsgReq := OpConMsgTypePLCJam;
	ELSIF tyOpConMsgReq = OpConMsgTypePLCJamStarted OR tyOpConMsgReq = OpConMsgTypePLCJam THEN
		tyOpConMsgReq := OpConMsgTypeNA;
		fbIdleTm (IN:= FALSE);
	ELSIF tyOpConMsgReq = OpConMsgTypePLCGrab THEN
		tyOpConMsgReq := OpConMsgTypeNA;
	ELSIF tyOpConMsgReq = OpConMsgTypePartProcessed THEN
		tyOpConMsgReq := OpConMsgTypeNA;
	ELSIF tyOpConMsgReq =  OpConMsgTypePartReceived THEN
		tyOpConMsgReq := OpConMsgTypeNA;
	END_IF

	//MsgReq (Event dependant)
	p_bPLCGrabPic := p_MCUL1StepPLCGrab OR p_MCUL2StepPLCGrab OR p_MCUL3StepPLCGrab;
	//PART PROCESSED ITEMS : [0-4], [progname, pitch, mag.type, mag.pos, mag.layer]
	tyPartProcessedItems.tyData.sValue[0] 	:= p_sLinkProdRcpCurrRcp1Nm;
	diTemp									:= p_diLinkProdRcpCurrRcp1Pitch;
	tyPartProcessedItems.tyData.sValue[1] 	:= DINT_TO_STRING(diTemp);
	tyPartProcessedItems.tyData.sValue[2] 	:= p_sLinkMagRcpCurrRcpNm;

	IF eOpsStep = TravLifULStepInitConv OR p_bPLCGrabPic THEN
		tyOpConMsgReq := OpConMsgTypePLCGrab;
		asMagEntered[1] := USINT_TO_STRING(BOOL_TO_USINT(p_bMagPresentSen1));
		asMagEntered[2] := USINT_TO_STRING(BOOL_TO_USINT(p_bMagPresentSen2));
		asMagEntered[3] := USINT_TO_STRING(BOOL_TO_USINT(p_bMagPresentSen3));
		IF p_bPLCGrabPic THEN
			bWaitMagChkRetCode := TRUE;
		END_IF
	ELSIF eOpsStep = TravLifULStepExitBrd THEN
		IF p_eLocalDSCommMod = McSetCommModSMEMA AND (p_eLocalDSSMEMAStatus = Done AND p_eLocalDSSMEMAStat = SMEMAActRun)
			AND (p_eConvStatus = Done AND p_eConvStat = ConvActExitPshr) THEN
			tyOpConMsgReq := OpConMsgTypePartProcessed;
			ELSIF (p_eLocalDSCommMod = McSetCommModHermes AND p_bLocalDSHermesStopTransport = FALSE)
			AND (p_eConvStatus = Done AND p_eConvStat = ConvActStopPshr) THEN
			tyOpConMsgReq := OpConMsgTypePartProcessed;
		END_IF
	ELSIF eOpsStep = TravLifULStepUSComm  THEN
		IF p_eConvStat = ConvActEnt THEN
			fbIdleTm (IN:= TRUE);
			IF fbIdleTm.Q THEN
				fbIdleTm (IN:= FALSE);
				bJamStarted := TRUE;
				tyOpConMsgReq := OpConMsgTypePLCJamStarted;
			END_IF
		END_IF
	ELSIF eOpsStep = TravLifULStepDSSigWait AND eGotoOpsStep = TravLifULStepTravLifMov THEN //transition
		//Magazine position  (pos )
		tyMagCoordinate.usiMagPos 					:=  UDINT_TO_USINT (udiPosAllwGo);
	ELSIF eOpsStep = TravLifULStepTravLifMov AND eGotoOpsStep = TravLifULStepDSSigRechk THEN //transition
		//Magazine layer  ( slot)
		IF p_bTopToBtm THEN
			IF eTravLifPosGo = 4 THEN
				diMagBrdQty[1] 				:=((ABS(p_diMaxSlt-p_diBuffer1NxtLoadSlt))/p_diLinkProdRcpCurrRcp1Pitch )+1;
				tyMagCoordinate.usiMagSlot 	:=  DINT_TO_USINT (diMagBrdQty[1]);
			ELSIF eTravLifPosGo = 5 THEN
				diMagBrdQty[2] 				:=((ABS(p_diMaxSlt-p_diBuffer2NxtLoadSlt))/p_diLinkProdRcpCurrRcp1Pitch )+1;
				tyMagCoordinate.usiMagSlot 	:=  DINT_TO_USINT (diMagBrdQty[2]);
			ELSIF eTravLifPosGo = 6 THEN
				diMagBrdQty[3] 				:=((ABS(p_diMaxSlt-p_diBuffer3NxtLoadSlt))/p_diLinkProdRcpCurrRcp1Pitch )+1;
				tyMagCoordinate.usiMagSlot 	:=  DINT_TO_USINT (diMagBrdQty[3]);
			END_IF
		ELSE  //btm to top
			IF eTravLifPosGo = 4 THEN
				diMagBrdQty[1] 				:=((ABS(p_diMinSlt-p_diBuffer1NxtLoadSlt))/p_diLinkProdRcpCurrRcp1Pitch )+1;
				tyMagCoordinate.usiMagSlot 	:=  DINT_TO_USINT (diMagBrdQty[1]);
			ELSIF eTravLifPosGo = 5 THEN
				diMagBrdQty[2] 				:=((ABS(p_diMinSlt-p_diBuffer2NxtLoadSlt))/p_diLinkProdRcpCurrRcp1Pitch )+1;
				tyMagCoordinate.usiMagSlot 	:=  DINT_TO_USINT (diMagBrdQty[2]);
			ELSIF eTravLifPosGo = 6 THEN
				diMagBrdQty[3] 				:=((ABS(p_diMinSlt-p_diBuffer3NxtLoadSlt))/p_diLinkProdRcpCurrRcp1Pitch )+1;
				tyMagCoordinate.usiMagSlot 	:=  DINT_TO_USINT (diMagBrdQty[3]);
			END_IF
		END_IF
		tyPartProcessedItems.tyData.sValue[3] 	:=  USINT_TO_STRING(tyMagCoordinate.usiMagPos);
		tyPartProcessedItems.tyData.sValue[4] 	:=  USINT_TO_STRING(tyMagCoordinate.usiMagSlot);
	ELSIF (eOpsStep =  TravLifULStepScanDS OR eOpsStep =  TravLifULStepHermesBCode) AND eGotoOpsStep = TravLifULStepWaitReturnCode THEN
		tyOpConMsgReq 	:= OpConMsgTypePartReceived;
	END_IF

	//Intterupting Event
	IF eGotoOpsStep <> eOpsStep THEN
		CASE eGotoOpsStep OF
			TravLifULStepTravLifMov:
				IF  bWaitMagChkRetCode AND eOpsStep <> TravLifULStepMagChkReturnCode AND eOpsStep <> TravLifULStepWaitReturnCode THEN
					eGotoOpsStep := TravLifULStepMagChkReturnCode;
				ELSIF p_bScanEn AND eOpsStep <> TravLifULStepWaitReturnCode THEN
					IF p_bConvHvBrd THEN
						eGotoOpsStep := TravLifULStepScanDS;
					END_IF
				ELSIF  eOpsStep <> TravLifULStepWaitReturnCode AND p_eLocalUSCommMod = McSetCommModHermes THEN
					IF p_bConvHvBrd THEN
						eGotoOpsStep := TravLifULStepHermesBCode;
					END_IF
				END_IF
		END_CASE
	END_IF
END_ACTION
```

#### Act_OpsScanner.st
```iecst
ACTION Act_OpsScanner:
	//DMC Scanner for Bosch
	//CASE
	bScannerEn := (p_tyNtParamDISettings.diScanComplSig <> 0 OR
	p_tyNtParamDOSettings.diScanTrigSig <> 0 ) AND p_bMcParamDMCScannerEn;
	bSignalTrigMagOutEn := (p_tyNtParamDOSettings.diMag1ExitPCB <> 0 OR
	p_tyNtParamDOSettings.diMag2ExitPCB <> 0 OR
	p_tyNtParamDOSettings.diMag3ExitPCB <> 0 ) AND p_bMcParamDMCScannerEn;
	bTCPScanner :=  (p_bTopScannerEn OR p_bBtmScannerEn);
	IF bScannerEn OR bSignalTrigMagOutEn OR bTCPScanner THEN
		CASE  eOpsStep OF
			TravLifULStepScanStdBy:
				bStartScanSig := TRUE;
				fbScanTimOut(IN:= TRUE,PT :=  DINT_TO_TIME(p_diMcParamDMCScanResponseTO));
				eTCPBtmAct   := TCPActFullWriteReadUntilValid*BOOL_TO_USINT(p_bBtmScannerEn);
				eTCPTopAct	 := TCPActFullWriteReadUntilValid*BOOL_TO_USINT(p_bTopScannerEn);
				IF (p_bDIPCBScanComplSig OR NOT(bScannerEn))
					AND
					(NOT(p_bBtmScannerEn) OR  (p_eTCPBtmStatus = Done AND p_eTCPBtmStat = TCPActFullWriteReadUntilValid ))
					AND
					(NOT(p_bTopScannerEn) OR  (p_eTCPTopStatus = Done AND p_eTCPTopStat = TCPActFullWriteReadUntilValid ))
					THEN //
					eTCPBtmAct := TCPActIdle_0*BOOL_TO_USINT(p_bBtmScannerEn);
					eTCPTopAct	 := TCPActIdle_0*BOOL_TO_USINT(p_bTopScannerEn);
					bStartScanSig := FALSE;
					eGotoOpsStep := TravLifULStepDSSigWait;
					fbScanTimOut(IN:= FALSE);
				ELSIF fbScanTimOut.Q THEN //Error
					bStartScanSig := FALSE;
					fbScanTimOut(IN:= FALSE);
					eStatus := Error;
					udiStatus	:= 10011;
				END_IF
		TravLifULStepExitBrd:
			IF bSignalTrigMagOutEn THEN
				IF eGotoOpsStep <> TravLifULStepExitBrd THEN
					bPCBExitMag1 := FALSE;
					bPCBExitMag2 := FALSE;
					bPCBExitMag3 := FALSE;
				ELSIF eTravLifPosGo = TravLifULPosDS1 THEN
					bPCBExitMag1 := TRUE;
				ELSIF eTravLifPosGo = TravLifULPosDS2 THEN
					bPCBExitMag2 := TRUE;
				ELSIF eTravLifPosGo = TravLifULPosDS3 THEN
					bPCBExitMag3 := TRUE;
				END_IF
			END_IF
		END_CASE

		//update in/output

		//interrupt (start scan)
		CASE  eGotoOpsStep OF
			TravLifULStepDSSigWait:
				IF eOpsStep <> TravLifULStepScanStdBy AND
					(eOpsStep = TravLifULStepInitTravLif OR eOpsStep = TravLifULStepEntBrd
					OR (eOpsStep = TravLifULStepInletPneuCls AND bSkipCloseInletShutter))
					AND (bScannerEn  ) THEN //temporary bypass
					eGotoOpsStep := TravLifULStepScanStdBy;
				END_IF

		END_CASE
	END_IF
END_ACTION
```
